(* Logix 5000 project; controller EuniceF_Lab1 vendor 1 type 14 code 150 rev 37.11; software revision 37.00 *)

TASK MainTask (continuous, watchdog 500 ms) : MainProgram

MODULES
   Local : vendor 1 type 14 code 150 (Compact 0, rev 37.11)
      Discrete_IO : Embedded (Compact 1, rev 3.1, Output RPI 20 ms)
      Analog_IO : Embedded (Compact 2, rev 1.1, Output RPI 80 ms)
      Counters : Embedded (Compact 3, rev 1.1, Output RPI 20 ms)
END_MODULES

VAR_GLOBAL   (* controller tags *)
   Countfor60cm : DINT;
   Default_Kfactor : DINT;
   Diif_Pressure : ALIAS FOR Local:2:O.Ch1Data;
   Done : ALIAS FOR Local:1:I.Data.15;
   Drain_Manual : ALIAS FOR Local:1:I.Data.4;
   DrainValve : ALIAS FOR Local:1:O.Data.10;
   Fill_Valve : ALIAS FOR Local:2:I.Ch1Data;
   Full : INT := 29208;
   Full_Btn : ALIAS FOR Local:1:I.Data.13;
   Good : ALIAS FOR Local:1:I.Data.14;
   Half : INT := -137;
   Half_Btn : ALIAS FOR Local:1:I.Data.12;
   HSC1_CurentCount : ALIAS FOR Local:3:I.Ctr0CurrentCount;
   K_factor : DINT;
   LevelMax : DINT;
   LevelMin : DINT;
   Mixer : ALIAS FOR Local:1:O.Data.9;
   Prove : BOOL;
   Pump : ALIAS FOR Local:1:O.Data.8;
   Quarter : INT := -15015;
   Quarter_Btn : ALIAS FOR Local:1:I.Data.11;
   Reset_HSC : ALIAS FOR Local:3:O.Ctr0SoftPreset;
   SEQ : DINT;
   Start : ALIAS FOR Local:1:I.Data.1;
   Status : STRING;
   Stop : ALIAS FOR Local:1:I.Data.2;
   T1 : TIMER := (PRE := 10000);
   Valve_Position : ALIAS FOR Local:2:O.Ch1Data;
   Zero : ALIAS FOR Local:1:I.Data.3;
END_VAR

PROGRAM MainProgram   (* main routine MainRoutine *)

ROUTINE MainRoutine   (* ladder *)
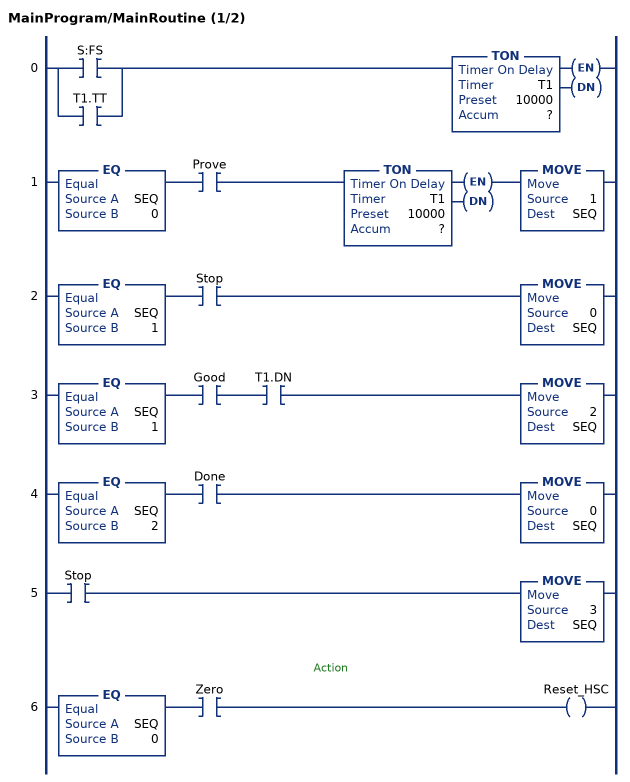
   0: [XIC(S:FS) ,XIC(T1.TT) ]TON(T1,?,?);
   1: EQ(SEQ,0)XIC(Prove)TON(T1,?,?)MOVE(1,SEQ);
   2: EQ(SEQ,1)XIC(Stop)MOVE(0,SEQ);
   3: EQ(SEQ,1)XIC(Good)XIC(T1.DN)MOVE(2,SEQ);
   4: EQ(SEQ,2)XIC(Done)MOVE(0,SEQ);
   5: XIC(Stop)MOVE(3,SEQ);
   // Action
   6: EQ(SEQ,0)XIC(Zero)OTE(Reset_HSC);
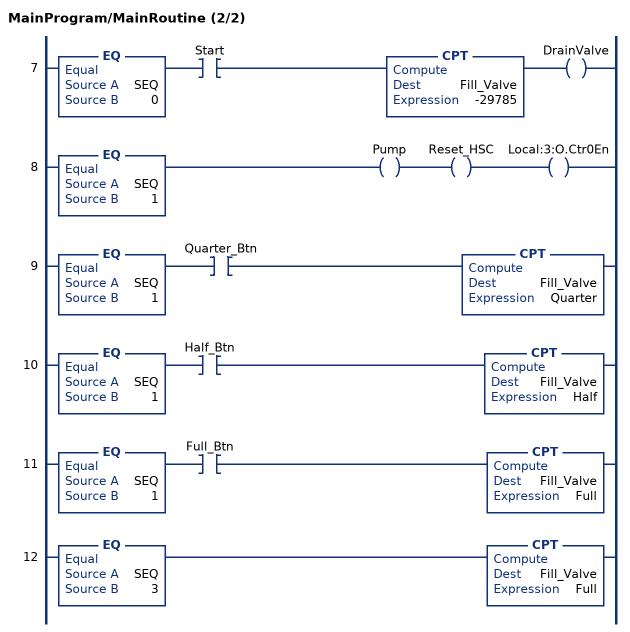
   7: EQ(SEQ,0)XIC(Start)CPT(Fill_Valve,-29785)OTE(DrainValve);
   8: EQ(SEQ,1)OTE(Pump)OTE(Reset_HSC)OTE(Local:3:O.Ctr0En);
   9: EQ(SEQ,1)XIC(Quarter_Btn)CPT(Fill_Valve,Quarter);
   10: EQ(SEQ,1)XIC(Half_Btn)CPT(Fill_Valve,Half);
   11: EQ(SEQ,1)XIC(Full_Btn)CPT(Fill_Valve,Full);
   12: EQ(SEQ,3)CPT(Fill_Valve,Full);
END_ROUTINE
END_PROGRAM
